// TIA Portal V20 export
DATA_BLOCK "BK10"   // DB306
// stored: MemoryReserve 100
   VAR
      "X10-1.ANODE FIX FRONT BACKWARD" : Bool := TRUE;
      "X11-1.SEPA CLAMP SAFETY PIN DETECT SENSOR" : Bool := FALSE;
      "X12-1.ANODE FIX REAR BACKWARD" : Bool := TRUE;
      "X13-1.SEPA CLAMP PRESSURE SWITCH" : Bool := FALSE;
      "X14-1.FIX ANODE DETECT SENSOR" : Bool := FALSE;
      "X15-1.SPARE" : Bool := FALSE;
      "X16-1.SPARE" : Bool := FALSE;
      "X17-1.SPARE" : Bool := FALSE;
      "X10-2.ANODE FIX FRONT FORWARD" : Bool := FALSE;
      "X11-2.SEPA GRIPPER SAFETY PIN DETECT SENSOR" : Bool := FALSE;
      "X12-2.ANODE FIX REAR FORWARD" : Bool := FALSE;
      "X13-2.SPARE" : Bool := FALSE;
      "X14-2.SPARE" : Bool := FALSE;
      "X15-2.SPARE" : Bool := FALSE;
      "X16-2.SPARE" : Bool := FALSE;
      "X17-2.SPARE" : Bool := FALSE;
   END_VAR
BEGIN
END_DATA_BLOCK
